# EPICS StreamDevice protocol: protocols/acq465.proto
Terminator = LF;
ExtraInput = Ignore;

acq465_fil_def {
	out "acq465_filter_default %d";
	in;
}

acq465_fil {
	out "acq465_filter %d";
	in;
}
